PROGRAM MC
VAR
	bMotorControlEnabled 	: BOOL := FALSE;
	iState					: INT := 0;
	sState					: WSTRING;
	tonAuxON				: TON;
	bEstopEngaged			: BOOL;
	tonDelay				: TON;
	tDelay					: TIME := T#5S;
	sAlarm					: WSTRING := " ";
	tReversing				: TIME;
	tForward				: TIME;
	bTimerOff				: BOOL := FALSE;
END_VAR

Inputs();

CASE iState OF
	0: sState := "E-Stop engaged";
			//HMI_IO.bDOStartLamp := FALSE;
			Module_IO.oStartLamp := FALSE;
			TS.oMotorON := FALSE;
			TS.oReverse := FALSE;
			TS.oForward := FALSE;
			tonDelay(IN:=FALSE);
	  	IF NOT bEstopEngaged THEN 
			sState := "E-Stop disengaged";
			IF Module_IO.iResetButton THEN 
				TS.oReset := TRUE;
				iState := 5;
	  		END_IF
		ELSE
			sState := "E-Stop engaged";
		END_IF
		IF Main.tonFlash.Q THEN
			//HMI_IO.bMCResetEstop := NOT HMI_IO.bMCResetEstop;
			Module_IO.oResetButton := NOT Module_IO.oResetButton;
		END_IF
		bTimerOff := FALSE;
	
	5:	sState := "Ready to Start Motor";
		TS.oReset := FALSE;
		bTimerOff := FALSE;
	    IF bMotorControlEnabled AND NOT bEstopEngaged THEN 
			tonDelay(IN:=FALSE);
			TS.oReverse := FALSE;
			TS.oForward := FALSE;
			//HMI_IO.bMCResetEstop := FALSE;
			Module_IO.oResetButton := FALSE;
			TS.oMotorON := FALSE;
			
			IF Main.tonFlash.Q THEN
				//HMI_IO.bDOStartLamp := NOT HMI_IO.bDOStartLamp;
				Module_IO.oStartLamp := NOT Module_IO.oStartLamp;
			END_IF
			IF Module_IO.iStartButton THEN
				iState := 10;
			END_IF
		ELSIF bEstopEngaged THEN
			iState := 0;
		END_IF
		
	10: sState := "Motor Forward/Reverse Control Enabled";
		TS.oMotorON := TRUE;
		Module_IO.oStartLamp := TRUE;
		tonDelay(IN:=FALSE);
		bTimerOff := FALSE;
		IF bMotorControlEnabled AND NOT bEstopEngaged THEN
			IF Module_IO.iForward THEN 
				iState := 20;
			ELSIF Module_IO.iReverse THEN
				iState := 30;
			END_IF
		ELSIF bEstopEngaged THEN
			iState := 0;
		ELSIF NOT bMotorControlEnabled THEN
			iState := 5;
		END_IF
		
	
	20: sState := "Running Forward";
		
		IF TS.oForward AND bMotorControlEnabled THEN
			bTimerOff := TRUE;
			tonDelay(IN:=Module_IO.iForward, PT:=tDelay, Q=>, ET=>tForward); //Safety when swtching the motor to reverse
			IF tonDelay.Q THEN 
				Module_IO.oForward := TRUE;
				//tonDelay(IN:=FALSE);
				bTimerOff := FALSE;
				(* tonAuxOn(IN:=TRUE, PT:=T#20S, Q=>, ET=>);
				IF Module_IO.iMotorContactorAux AND NOT tonAuxOn.Q THEN 
					tonAuxON(IN:=FALSE);
				ELSE
					sAlarm := "Forward Control issue, Press Emergency Stop";
					Module_IO.oForward := FALSE;
					iState := 100;
				END_IF  *)
			END_IF
		ELSE 
			Module_IO.oForward := FALSE;
			tonDelay(IN:=FALSE);
			iState := 10;
		END_IF
		IF NOT bMotorControlEnabled THEN
			iState := 5;
		ELSIF bEstopEngaged THEN
			iState := 0;
		END_IF
		
	30: sState := "Running Reverse";
	
		IF TS.oReverse AND bMotorControlEnabled THEN
			bTimerOff := TRUE;
			tonDelay(IN:=Module_IO.iReverse, PT:=tDelay, Q=>, ET=>tReversing); //Safety when swtching the motor to reverse
			IF tonDelay.Q THEN 
				Module_IO.oReverse := TRUE;
				//tonDelay(IN:=FALSE);
				bTimerOff := FALSE;
				(*tonAuxOn(IN:=TRUE, PT:=T#20S, Q=>, ET=>);
				IF Module_IO.iMotorContactorAux AND NOT tonAuxOn.Q THEN 
					tonAuxON(IN:=FALSE);
				ELSE
					sAlarm := "Reverser Control issue, Press Emergency Stop";
					Module_IO.oForward := FALSE;
					iState := 100;
				END_IF *)
			END_IF
		ELSE 
			Module_IO.oReverse := FALSE;
			tonDelay(IN:=FALSE);
			iState := 10;
		END_IF
		IF NOT bMotorControlEnabled THEN
			iState := 5;
		ELSIF bEstopEngaged THEN
			iState := 0;
		END_IF
		
    100: 
		sState := "Alarm: {sALARM}";
		TS.oMotorON := FALSE;
		bTimerOff := FALSE;
		Module_IO.oStartLamp := FALSE;
		IF Main.tonFlash.Q THEN
			//HMI_IO.bMCResetEstop := NOT HMI_IO.bMCResetEstop;
			Module_IO.oResetButton := NOT Module_IO.oResetButton;
		END_IF
	
END_CASE

//First thing to check in case motor is not running
bMotorControlEnabled := Module_IO.iStopButton;// AND NOT Module_IO.iMotorOverLoad;
bEstopEngaged := NOT TS.iEStop1 OR NOT TS.iEStop2;
TS.oOverload := FALSE; //Indicator Only

ACTION Inputs:
//From Twinsafe

TS.oForward := Module_IO.iForward;
TS.oReverse := Module_IO.iReverse;

Module_IO.oForward := TS.iForward;
Module_IO.oReverse := TS.iReverse;

//TS.oContactor := Module_IO.iMotorContactorAux;
TS.oOverload := Module_IO.iMotorOverLoad;
END_ACTION

END_PROGRAM

(* stored: Version 1.1.0.1, ProductVersion 3.1.4024.11
   POU MC: Id {809264f6-585b-4a63-b4a9-f649718cd946}, SpecialFunc None
   Action Inputs: Id {3d897027-50b9-4c10-8557-88afed10ddf6} *)
